PROGRAM Homing
VAR
	
END_VAR

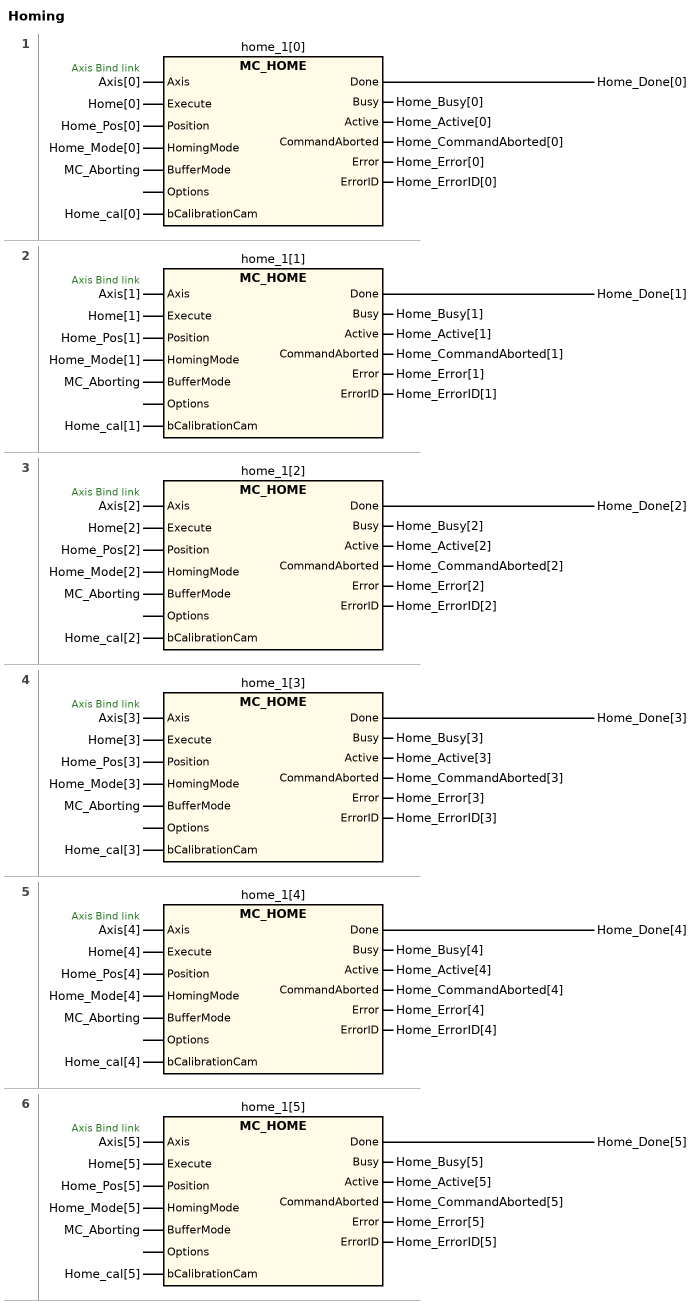
// NETWORK 1
//   home_1[0]: HOME
//   Axis[0]: Axis Bind link
home_1[0](
    Axis := Axis[0],
    Execute := Home[0],
    Position := Home_Pos[0],
    HomingMode := Home_Mode[0],
    BufferMode := MC_Aborting,
    bCalibrationCam := Home_cal[0],
    Busy => Home_Busy[0],
    Active => Home_Active[0],
    CommandAborted => Home_CommandAborted[0],
    Error => Home_Error[0],
    ErrorID => Home_ErrorID[0]); // MC_HOME
Home_Done[0] := home_1[0].Done;

// NETWORK 2
//   home_1[1]: HOME
//   Axis[1]: Axis Bind link
home_1[1](
    Axis := Axis[1],
    Execute := Home[1],
    Position := Home_Pos[1],
    HomingMode := Home_Mode[1],
    BufferMode := MC_Aborting,
    bCalibrationCam := Home_cal[1],
    Busy => Home_Busy[1],
    Active => Home_Active[1],
    CommandAborted => Home_CommandAborted[1],
    Error => Home_Error[1],
    ErrorID => Home_ErrorID[1]); // MC_HOME
Home_Done[1] := home_1[1].Done;

// NETWORK 3
//   home_1[2]: HOME
//   Axis[2]: Axis Bind link
home_1[2](
    Axis := Axis[2],
    Execute := Home[2],
    Position := Home_Pos[2],
    HomingMode := Home_Mode[2],
    BufferMode := MC_Aborting,
    bCalibrationCam := Home_cal[2],
    Busy => Home_Busy[2],
    Active => Home_Active[2],
    CommandAborted => Home_CommandAborted[2],
    Error => Home_Error[2],
    ErrorID => Home_ErrorID[2]); // MC_HOME
Home_Done[2] := home_1[2].Done;

// NETWORK 4
//   home_1[3]: HOME
//   Axis[3]: Axis Bind link
home_1[3](
    Axis := Axis[3],
    Execute := Home[3],
    Position := Home_Pos[3],
    HomingMode := Home_Mode[3],
    BufferMode := MC_Aborting,
    bCalibrationCam := Home_cal[3],
    Busy => Home_Busy[3],
    Active => Home_Active[3],
    CommandAborted => Home_CommandAborted[3],
    Error => Home_Error[3],
    ErrorID => Home_ErrorID[3]); // MC_HOME
Home_Done[3] := home_1[3].Done;

// NETWORK 5
//   home_1[4]: HOME
//   Axis[4]: Axis Bind link
home_1[4](
    Axis := Axis[4],
    Execute := Home[4],
    Position := Home_Pos[4],
    HomingMode := Home_Mode[4],
    BufferMode := MC_Aborting,
    bCalibrationCam := Home_cal[4],
    Busy => Home_Busy[4],
    Active => Home_Active[4],
    CommandAborted => Home_CommandAborted[4],
    Error => Home_Error[4],
    ErrorID => Home_ErrorID[4]); // MC_HOME
Home_Done[4] := home_1[4].Done;

// NETWORK 6
//   home_1[5]: HOME
//   Axis[5]: Axis Bind link
home_1[5](
    Axis := Axis[5],
    Execute := Home[5],
    Position := Home_Pos[5],
    HomingMode := Home_Mode[5],
    BufferMode := MC_Aborting,
    bCalibrationCam := Home_cal[5],
    Busy => Home_Busy[5],
    Active => Home_Active[5],
    CommandAborted => Home_CommandAborted[5],
    Error => Home_Error[5],
    ErrorID => Home_ErrorID[5]); // MC_HOME
Home_Done[5] := home_1[5].Done;

END_PROGRAM

(* stored: Version 1.1.0.1, ProductVersion 3.1.4018.5
   POU Homing: Id {f643a52b-e5c8-4310-a463-8235f37d8938}, SpecialFunc None *)
